INTERFACE ITF_Cylinder EXTENDS __System.IQueryInterface

PROPERTY AtHome : bool
GET
END_GET
END_PROPERTY

PROPERTY AtWork : bool
GET
END_GET
END_PROPERTY

METHOD MoveToHome
VAR_INPUT
END_VAR
END_METHOD

METHOD MoveToWork
VAR_INPUT
END_VAR
END_METHOD

PROPERTY MovingToHomePosition : BOOL
GET
END_GET
END_PROPERTY

PROPERTY MovingToWorkPosition : BOOL
GET
END_GET
END_PROPERTY

END_INTERFACE

(* stored: Version 1.1.0.1, ProductVersion 3.1.4024.4
   Itf ITF_Cylinder: Id {d67e700f-f4ae-4803-bb24-213c42f7b180}
   Property AtHome: Id {de61584f-b4cf-4cc1-9dae-bfa15f41af2a}
   Get Get: Id {dee60c83-dbdf-4df2-9d01-cb15f4a035a3}
   Property AtWork: Id {86608e1a-db36-448a-ab9b-c98dba75f077}
   Get Get: Id {c885c12e-772c-4067-b1a8-f3eeab530dd2}
   Method MoveToHome: Id {8e4809ef-bb6b-4b80-ac93-e8ed0d61f227}
   Method MoveToWork: Id {ea959bff-fd62-4b67-bd52-9c1b6742dba9}
   Property MovingToHomePosition: Id {8f8db5f6-af30-4702-922c-4dc6e7e162f2}
   Get Get: Id {58b7f0d7-6c80-4cf3-ac2e-e745891ad9a0}
   Property MovingToWorkPosition: Id {5b9b1d60-96c5-41a3-961c-d8cc7c58d34c}
   Get Get: Id {ce3660d6-fde2-4739-aebd-0e703ab1f59b} *)
